TYPE stBS02PL_Line EXTENDS stPIM_LineEventsModule :
STRUCT

	{attribute 'OPC.UA.DA' := '1'}
	stStation_BS02PL01 : stPIM_StationEventsModule_1_Machine;
END_STRUCT
END_TYPE

(* stored: Version 1.1.0.1, ProductVersion 3.1.4024.15
   DUT stBS02PL_Line: Id {2274495f-863b-4862-ae42-86dde84efdee} *)
